{attribute 'qualified_only'}
{attribute 'strict'}
{attribute 'to_string'}
TYPE E_VisionMode :
(
    Simulation := 0,
    Camera     := 10
);
END_TYPE

(* stored: Version 1.1.0.1, ProductVersion 3.1.4026.20
   DUT E_VisionMode: Id {64E298A0-87A1-41AD-B6F2-53D818CB89F6} *)
